PROGRAM Main
VAR
	// Standalone command execution
	pStandaloneCommand : POINTER TO DummyCommand;
	runStandaloneCommand : BOOL;
	abortStandaloneCommand : BOOL;
	simulateErrorStandaloneCommand : BOOL;
	simulatedStandaloneCommandErrorId : UDINT := 1234;
	
	standaloneCommandResult : I_Result;
	standaloneCommandCompleted : BOOL;
	standaloneCommandAborted : BOOL;
	standaloneCommandError : BOOL;
	standaloneCommandErrorId : UDINT;
	
	// SingleAsyncCommandRunner command execution
	
	// QueuedPoolAsyncCommandRunner command execution
	runQueuedPoolCommand : BOOL;
	pQueuedCommand : POINTER TO DummyCommand;

	queuedPoolCommandRunner : QueuedPoolAsyncCommandRunner(poolCapacity := 2, queueCapacity := 5);
	
	// Support variables
	id : DINT;
END_VAR

// Standalone command execution
IF runStandaloneCommand THEN
	runStandaloneCommand := FALSE;
	pStandaloneCommand := __NEW(DummyCommand(id := NextId(), name := 'standalone'));
END_IF

IF pStandaloneCommand <> 0 THEN
	IF pStandaloneCommand^.Idle THEN
		pStandaloneCommand^.Execute();
	ELSIF pStandaloneCommand^.Executing THEN
		pStandaloneCommand^.CyclicCall();
		
		IF abortStandaloneCommand THEN
			abortStandaloneCommand := FALSE;
			pStandaloneCommand^.Abort();
		END_IF
		
		IF simulateErrorStandaloneCommand THEN
			simulateErrorStandaloneCommand := FALSE;
			pStandaloneCommand^.SimulateError(simulatedStandaloneCommandErrorId);
		END_IF
	ELSIF pStandaloneCommand^.Stopped THEN
		standaloneCommandResult := pStandaloneCommand^.GetResult();
		__DELETE(pStandaloneCommand);
		standaloneCommandCompleted := standaloneCommandResult.Completed;
		standaloneCommandAborted := standaloneCommandResult.Aborted;
		standaloneCommandError := standaloneCommandResult.Error;
		standaloneCommandErrorId := standaloneCommandResult.ErrorId;
		standaloneCommandResult.Dispose();
		standaloneCommandResult := 0;
	END_IF
END_IF

// SingleAsyncCommandRunner command execution

// QueuedPoolAsyncCommandRunner command execution
IF runQueuedPoolCommand THEN
	runQueuedPoolCommand := FALSE;
	pQueuedCommand := __NEW(DummyCommand(id := NextId(), name := 'queued-pool'));
	queuedPoolCommandRunner.QueueCommand(pQueuedCommand^);
END_IF

queuedPoolCommandRunner.CyclicCall();

METHOD PRIVATE NextId : DINT
NextId := id;
id := id + 1;
END_METHOD

END_PROGRAM

(* stored: Version 1.1.0.1, ProductVersion 3.1.4026.6
   POU Main: Id {ca1e1f26-6d15-4483-9500-7f4e2de7b73c}, SpecialFunc None
   Method NextId: Id {f4c2d668-26f2-4c78-b288-a09ab44f096f} *)
